FUNCTION TryConvert_WORD_TO_UDINT : BOOL
VAR_INPUT
	in : WORD;
	out : REFERENCE TO UDINT;
END_VAR

out := WORD_TO_UDINT(in);
TryConvert_WORD_TO_UDINT := TRUE;

END_FUNCTION

(* stored: Version 1.1.0.1, ProductVersion 3.1.4024.12
   POU TryConvert_WORD_TO_UDINT: Id {392bf19c-f63f-46f2-8edb-9fc6e20840a9}, SpecialFunc None *)
